// TwinCAT 3 PLC project PLC
// ProgramVersion: 3.1.4026.19
// CompilerDefines: VISU_USEPROPERTYINFO
// libraries:
//   Tc2_Standard, * (Beckhoff Automation GmbH)
//   Tc2_System, * (Beckhoff Automation GmbH)
// project tree:
//   / GlobalTextList.TcGTLO, PlcTask.TcTTO, Visualization Manager.TcVMO (not stored)
//   POUs/ MAIN.TcPOU
//   VISUs/ Visualization.TcVIS
// real-time tasks:
//   TASK PlcTask: cycle T#10ms, priority 20, ADS port 350

CONFIGURATION PLC
    RESOURCE PLC ON TwinCAT3
        TASK PlcTask(INTERVAL := T#10ms, PRIORITY := 20);
        PROGRAM MAIN WITH PlcTask : MAIN;
    END_RESOURCE
END_CONFIGURATION

// ---- POUs/MAIN.TcPOU
PROGRAM MAIN
VAR
	bStartButton : BOOL;
	bStopButton : BOOL;
	
	bSystemActive : BOOL;
	
	bHorn : BOOL;
	bMotor : BOOL;
	
	fbStartupTimer : TON;
END_VAR

IF bStopButton THEN
	bSystemActive := FALSE;

ELSIF bStartButton THEN
	bSystemActive := TRUE;
END_IF

fbStartupTimer(IN := bSystemActive, PT := T#5S);

bHorn := bSystemActive AND NOT fbStartupTimer.Q;

bMotor := bSystemActive AND fbStartupTimer.Q;

END_PROGRAM

// ---- GlobalTextList.TcGTLO
TEXTLIST GlobalTextList
  981 = 'Horn'
  52 = 'Motor'
  372 = 'Time: %s'
END_TEXTLIST

// ---- VISUs/Visualization.TcVIS
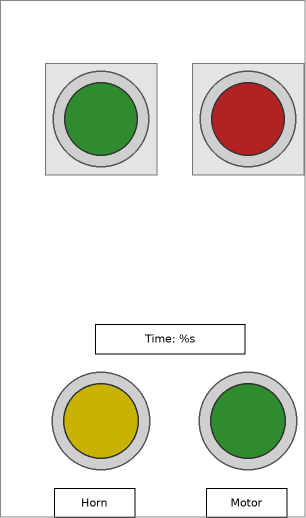
VISUALIZATION Visualization  // 306x518
    PushSwitch (43,63 116x112), variable: MAIN.bStartButton, behaviour: TOGGLE, style: Switch-PushSwitch-Green
    PushSwitch (190,63 116x112), variable: MAIN.bStopButton, behaviour: TOGGLE, style: Switch-PushSwitch-Red
    Lamp1 (43,364 116x114), variable: MAIN.bHorn, style: Lamp-Lamp1-Yellow
    Lamp1 (190,364 116x114), variable: MAIN.bMotor, style: Lamp-Lamp1-Green
    Rectangle (95,324 150x30), "Time: %s", text variable: MAIN.fbStartupTimer.ET
    Rectangle (54,488 81x30), "Horn", text variable: MAIN.fbStartupTimer.ET
    Rectangle (206,488 81x30), "Motor", text variable: MAIN.fbStartupTimer.ET
END_VISUALIZATION
